Staubli VAL3: buildList.pgx

program buildList()
  local num l_nSize
  local string l_sEvent
  local num i
  local bool l_bFound
  local num l_nCount
  local string l_sEmpty
  local num j
begin
    call use:stringCopy(l_sEmpty,sList)
  ////  call use:setSizeList(17,0,21,7)
  ////  call use:setSizeList(15,0,18,9)
  ////  建立对话款
  ////  call use:listcreate("")

  //  sWorkingmode[0]="[ ] 生产循环状态"
  //  sWorkingmode[1]="[ ] 循环暂停状态"
  //  sWorkingmode[2]="[ ] 机器人HOME点"
  //  sWorkingmode[3]="[ ] 机器人准备好"
  //  sWorkingmode[4]="[ ] 急停报警"
  //  sWorkingmode[5]="[ ] 防止碰撞功能开启"
  //  sWorkingmode[6]="[ ] 通讯正常"

  //  call use:listadd(sWorkingmode)
  //  call use:selectNewField(nSelected,nIndex,nView)
  //  call use:listupdate(0)
  // nIndex=data:nPage_Traj
  // call use:selectNewField(nSelected,nIndex,nView)
end
